PROGRAM MAIN
VAR
END_VAR

END_PROGRAM

(* stored: Version 1.1.0.1
   POU MAIN: Id {4e56a9cf-11b3-422e-b81c-eb6828dd29be} *)
